(* CoDeSys 2.3 export: VISUPORTESET3.EXP *)

(* POU Simulation_Visuelle/VisuPortesET3, ST *)
FUNCTION VisuPortesET3 : BOOL
VAR_INPUT
END_VAR
VAR
	TimerDeTempo: TP;
	CompteurPortesVisu: INT;
	CompteurVarVisu: INT;
	CompteurDeTemps: INT;
	Step: INT;
	CompteurLocal: INT;
	CONTACTEUR_SEC: INT;
END_VAR
(* Cette fonction sert à fermer les portes de l'etage 3 en fonction des donné transmises par le porgramme principal*

	La fonction va simuler une fermeture sur action d'un moteur, et simuler le capteur  lorsque la coordonée de position fermé est atteinte : x=0 et y=-2*)
IF F3 OR O3 THEN
	(*On simule la position physique du contacteur avec des coordonnées*)
	IF F3 THEN CONTACTEUR_SEC:=-71;
	ELSE CONTACTEUR_SEC:=0;END_IF
	wait(IN:=TRUE, PT:=T#1ms);
	FOR CompteurLocal:=1 TO 3 BY 1 DO
		IF NOT wait.Q THEN
			wait(IN:=FALSE);
			(* en fonction de l'état du contacteur nous allons
			simuler une ouverture/fermeture de la porte*)

			(* nous allons utiliser les fonctions de coordonnées
			pour que la simulation suivent une trajectoire excate et soienet parfaitement synchronisé*)
			IF VisuET3Dx > CONTACTEUR_SEC THEN
				VisuET3Dx:=VisuET3Dx-1;
				VisuET3Dy:=FX_PorteD(VisuET3Dx);
				VisuET3Gx:=FX_Porte_Vitesse(VisuET3Dx);
				VisuET3Gy:=FX_PorteG(VisuET3Gx);
			ELSIF  VisuET3Dx < CONTACTEUR_SEC THEN
				VisuET3Dx:=VisuET3Dx+1;
				VisuET3Dy:=FX_PorteD(VisuET3Dx);
				VisuET3Gx:=FX_Porte_Vitesse(VisuET3Dx);
				VisuET3Gy:=FX_PorteG(VisuET3Gx);
			END_IF
		END_IF
	END_FOR
END_IF

IF VisuET3Dx = - 71  THEN P3fer:=TRUE;
ELSE P3fer:=FALSE;END_IF

IF VisuET3Dx = 0  THEN P3ouv:=TRUE;
ELSE P3ouv:=FALSE;END_IF
END_FUNCTION
